Xinje XDPPro project, PLC1: XDME-60T10 (software 3.7.14b 2022-06-24)

PROGRAM 梯形图

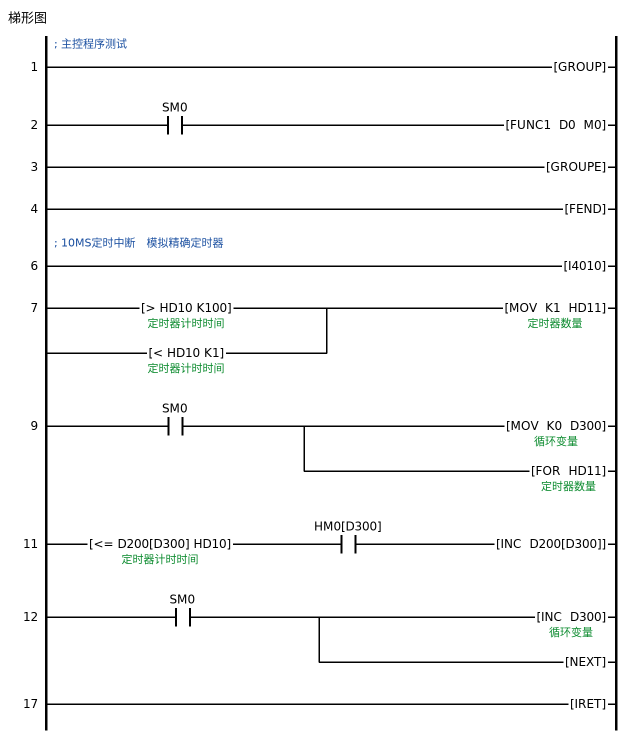
; 主控程序测试
GROUP
LD     SM0
FUNC1  D0 M0
GROUPE
FEND
; 10MS定时中断　模拟精确定时器
I4010
LD>    HD10 K100	; 定时器计时时间
OR<    HD10 K1	; 定时器计时时间
MOV    K1 HD11	; 定时器数量
LD     SM0
MOV    K0 D300	; 循环变量
FOR    HD11	; 定时器数量
LD<=   D200[D300] HD10	; 定时器计时时间
AND    HM0[D300]
INC    D200[D300]
LD     SM0
INC    D300	; 循环变量
NEXT
IRET

COMMENTS (devices not used above)
D200	定时器1
HM0	定时器开启标志

C FUNCTION BLOCK func1.fcb
/* C语言常用技术要点
#EXPORT_ENTRY_BEGIN(FUNC1)
//    类型              模式             个数               映射          注释
W = { type = "PINT16S", mode = [In,Out], count = "unknown", map = [D,HD], comment = "" }
B = { type = "BIT"    , mode = [In,Out], count = "unknown", map = [M,HM], comment = "" }
#EXPORT_ENTRY_END */
/*************************************************************************
 * FunctionBlockName:  FUNC1
 * Version:            1.0.0
 * Author:             LittleWhite
 * UpdateTime:         2022-07-25 16:53:27
 * Comment:            C语言常用技术要点
**************************************************************************/

/**
 * @summary
 * @param W
 * @param B
 */
#include "func1.h"
void FUNC1 ( PINT16S W, BIT B )
{
#define SysRegAddr_HD_D_HM_M





    /***************宏定义使用*********************/
    Car_Total = 100;
    Grid_Total = 100;
    Speed_Average = 2.0;

    TimerNumbers = 100;             //定时器数量设置
    TimerLimit = 100;               //定时器时间限制 单位:10ms

    //这里是不会检查类型是否匹配，以及内村溢出等问题的
    /***************使用条码结构体组*********************/
    Code_Info *pCode_Info[5];                        //定义5个条码组成的结构体组
    for ( int i = 0; i < 5; i++ )
    {
        pCode_Info[i] = ( Code_Info * ) ( Pack_Code_First_Address + i * sizeof ( Code_Info ) / 2 ); //指针指向储存区域
    }  
    

    pCode_Info[0]->Length = 1;
    pCode_Info[0]->Character[0] = 'a';

    pCode_Info[1]->Length = 1;
    pCode_Info[1]->Character[0] = 'b';

    pCode_Info[2]->Length = 1;
    pCode_Info[2]->Character[0] = 'c';

    pCode_Info[3]->Length = 1;
    pCode_Info[3]->Character[0] = 'd';

    pCode_Info[4]->Length = 1;
    pCode_Info[4]->Character[0] = 'e';


    /**********************字符串的使用**********************/
    char *p;
    p = ( char * ) ( Sorting_Grid_First_Address );
    char str[] = "123213";
    for ( int i = 0; i < sizeof ( str ); i++ )
    {
        * ( p + i )  = str[i];
    }
    
//#define TimerValueArray                             (&D[200])          //模拟精确定时器1-100 D[200]-D[399]
//#define TimerTriggerArray                           (&D[400])          //定时器触发次数1-100 D[400]-D[499]
    //这里是一个数据寄存器‘D’ 存储一个字符（char）嘛？

    /**********************定时器到达设定时间复位**********************/
    for ( int i = 0; i < 100; i++ )
    {
        if ( TimerValueArray[i] >= TimerLimit )
        {
            TimerValueArray[i] = 0;
            TimerTriggerArray[i] = TimerTriggerArray[i] + 1;
        }
    }
}

C FILE func1.h
#ifndef	_FUNC1_H
#define	_FUNC1_H

/*类似于一种强制类型转换的引用做法?，不对 宏定义并不做任何处理，只是将宏的内容展开，所以后面加上中括号的情况应该直接加在这个式子尾部去看*/
#define DHD   *(INT32S*)&HD    //32位有符号整形
#define FHD   *(FP32*)&HD    //32位浮点型
#define DSD   *(INT32S*)&SD
#define FSD   *(FP32*)&SD
#define DHSD  *(INT32S*)&HSD
#define DHSCD *(INT32S*)&HSCD
#define D_D	     *(INT32S*)&D
#define F_D      *(FP32*)&D
#pragma pack(2)

  
/************************寄存器可以直接通过宏定义操作使用******************************/
#define Car_Total                                       HD[0]             //小车总数
#define Grid_Total                                      HD[1]             //格口总数
#define Speed_Average                                   FHD[2]            //环线速度 浮点 单位m/s
#define TimerLimit                                      HD[10]            //定时器计时时间
#define TimerNumbers                                    HD[11]            //定时器数量  最大100个
/********************错误定义方法************************/
//#define ErrorDefine1                                     FHD[3]            //双字占用禁用奇数1    
//#define ErrorDefine2                                     DHD[5]            //双字占用禁用奇数2       

/************************M寄存器不能直接进行宏定义******************************/
/*****************为什么呢 难道是类似于临时变量 宏定义之后也没有作用吗*****************/
//#define Mark                                               M[0]          //不能如此使用

/****************  分拣格口定义  ************************/
typedef struct
{
    INT16U TargetGridNumbers;         //上位机分配格口数量
    INT16U TargetGrid[7];             //分配的格口号
} Sorting_Grid;
/****************  包裹单号/序列号信息  ************************/
typedef struct
{
    INT16U Length;                  //单号/序列号长度
    INT8U  Character[22];           //最长22位单号或者22位序列号
    INT16U Expand[8];               //扩展8个字
} Code_Info;
#define Sorting_Grid_First_Address                  D+0                //分拣格口存储
#define Pack_Code_First_Address                     D+100              //包裹条码存储
#define TimerValueArray                             (&D[200])          //模拟精确定时器1-100 D[200]-D[399]
#define TimerTriggerArray                           (&D[400])          //定时器触发次数1-100 D[400]-D[499]


/*******************新增部分*****************/
#define Car_Mark                                    D[999]              //小车号
#define 

#endif